// Mitsubishi GX Works2 project: 시퀀스 부분 반복 회로 (카운터-시퀀스 유지)   PLC: Q03UDV

PROGRAM MAIN
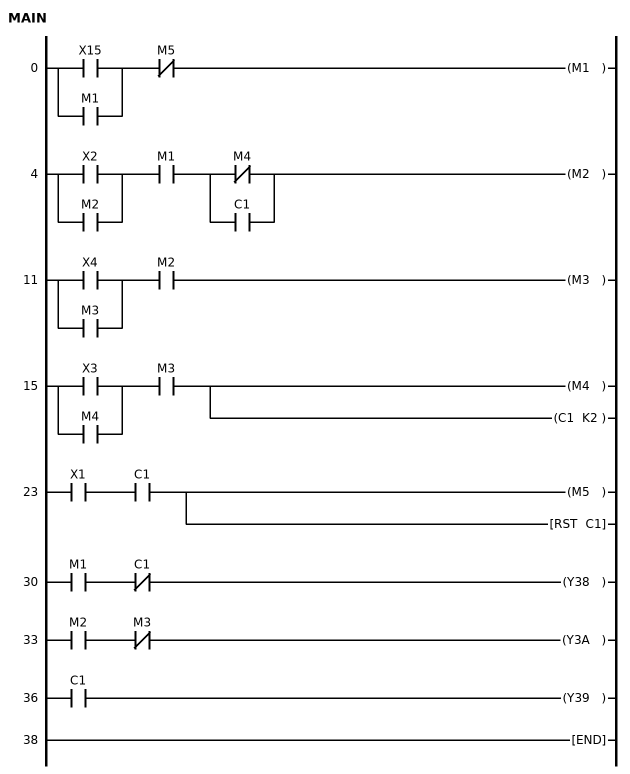
0     LD      X15
      OR      M1
      ANI     M5
      OUT     M1
4     LD      X2
      OR      M2
      AND     M1
      LDI     M4
      OR      C1
      ANB
      OUT     M2
11    LD      X4
      OR      M3
      AND     M2
      OUT     M3
15    LD      X3
      OR      M4
      AND     M3
      OUT     M4
      OUT     C1 K2
23    LD      X1
      AND     C1
      OUT     M5
      RST     C1
30    LD      M1
      ANI     C1
      OUT     Y38
33    LD      M2
      ANI     M3
      OUT     Y3A
36    LD      C1
      OUT     Y39
38    END
END_PROGRAM
